FUNCTION_BLOCK FB_BUTTON
VAR_INPUT
	///Pointer Button-Variable
	pbtIN: POINTER TO structButton;
	///Button disable
	xINdis: BOOL;
	///Anzeige Grün
	xINon: BOOL;
	///Anzeige Rot
	xINerr: BOOL;
END_VAR
VAR
	rt: R_TRIG;
	ft: F_TRIG;
END_VAR

pbtIN^.disable := xINdis;
IF pbtIN^.disable THEN
	pbtIN^.button := FALSE;
END_IF
pbtIN^.press := pbtIN^.button AND NOT pbtIN^.disable;
rt(CLK:= pbtIN^.press, Q=> pbtIN^.rtrig);
ft(CLK:= pbtIN^.press, Q=> pbtIN^.ftrig);
pbtIN^.on := xINon;
pbtIN^.error := xINerr;

END_FUNCTION_BLOCK

(* stored: Version 1.1.0.1, ProductVersion 3.1.4024.6
   POU FB_BUTTON: Id {e094881a-1744-42f9-9039-9031cce944e2}, SpecialFunc None *)
